// TwinCAT 3 PLC project MachineAlarmManager
// Title: machine_alarm_manager
// Company: Beckhoff Automation K.K.
// Author: Takashi Ichihashi
// ProjectVersion: 1.0.2.0
// ProgramVersion: 3.1.4024.0
// CompilerDefines: VISU_USEWSTRING
// libraries:
//   Tc2_Standard, * (Beckhoff Automation GmbH)
//   Tc2_System, * (Beckhoff Automation GmbH)
//   Tc2_Utilities, * (Beckhoff Automation GmbH)
//   Tc3_EventLogger, * (Beckhoff Automation GmbH)
//   Tc3_Module, * (Beckhoff Automation GmbH)
//   VisuSymbols,3.5.10.0,System
// project tree:
//   DUTs/ AlarmMessage.TcDUT, EventContainer.TcDUT, DataTag.TcDUT, EventActivityFields.TcDUT, EventQueueCommand.TcDUT, EventSeverityStatusMember.TcDUT, EventText.TcDUT, primitives.TcDUT, ST_EventMetadata.TcDUT, ST_EventView.TcDUT, Tc2EventClass.TcDUT, Tc2EventStates.TcDUT
//   / GlobalTextList.TcGTLO, PlcTask.TcTTO, Visualization Manager.TcVMO (not stored), VISU_TASK.TcTTO
//   GVLs/ AlarmEventParam.TcGVL, GVL.TcGVL
//   POUs/ FB_Alarm.TcPOU, FB_EventIoTExporter.TcPOU, FB_EventObserver.TcPOU, FB_Subject.TcPOU, FB_TcEventQueue.TcPOU, FB_Tc3EventVisualizationView.TcPOU, FB_TcEventTable.TcPOU, InterfaceEventViewer.TcIO, AlarmManager.TcPOU, MAIN.TcPOU, UserProgram.TcPOU
//   VISUs/ languages.TcTLO, Visualization.TcVIS, history.TcVIS, current.TcVIS
// real-time tasks:
//   TASK PlcTask: cycle T#10ms, priority 20, ADS port 350
//   TASK VISU_TASK: cycle T#200000us, priority 30, ADS port 351

CONFIGURATION MachineAlarmManager
    RESOURCE PLC ON TwinCAT3
        TASK PlcTask(INTERVAL := T#10ms, PRIORITY := 20);
        TASK VISU_TASK(INTERVAL := T#200000us, PRIORITY := 30);
        PROGRAM MAIN WITH PlcTask : MAIN;
        PROGRAM VisuElems_Visu_Prg WITH VISU_TASK : VisuElems.Visu_Prg;
    END_RESOURCE
END_CONFIGURATION

// ---- DUTs/AlarmMessage.TcDUT
TYPE AlarmMessage EXTENDS EventActivityFields :
STRUCT
	datetime: ULINT;
	sequence_number: ULINT;
END_STRUCT
END_TYPE

// ---- DUTs/EventContainer.TcDUT
TYPE EventContainer :
STRUCT
	event : FB_Alarm;
	{attribute 'TcEncoding' := 'UTF-8'}
	event_text	: T_MaxString;
END_STRUCT
END_TYPE

// ---- DUTs/DataTag.TcDUT
TYPE DataTag :
STRUCT
	{attribute 'TagName' := 'machine_id'}
    machine_id : STRING;
	{attribute 'TagName' := 'module_name'}
    module_name: STRING;
END_STRUCT
END_TYPE

// ---- DUTs/EventActivityFields.TcDUT
TYPE EventActivityFields EXTENDS DataTag:
STRUCT
	{attribute 'TagName' := 'uuid'}
    uuid : STRING;
	{attribute 'FieldName' := 'event_id'}
    event_id : STRING;
	{attribute 'FieldName' := 'severity'}
	severity: INT;
	{attribute 'TcEncoding' := 'UTF-8'}
	{attribute 'FieldName' := 'text'}
    text : STRING;
	{attribute 'FieldName' := 'status'}
    status : BOOL;
END_STRUCT
END_TYPE

// ---- DUTs/EventQueueCommand.TcDUT
TYPE EventQueueCommand :
STRUCT
	metadata : ST_EventMetadata;
	event_text_processor	: FB_RequestEventText;
	event_details_processor	: FB_RequestEventDetails;
END_STRUCT
END_TYPE

// ---- DUTs/EventSeverityStatusMember.TcDUT
TYPE EventSeverityStatusMember :
STRUCT
	severity 	: TcEventSeverity;
	active_counter		: UINT;
	raised_counter		: UINT;
	confirmed_counter	: UINT;
END_STRUCT
END_TYPE

// ---- DUTs/EventText.TcDUT
TYPE EventText :
STRUCT
	event : I_TcEventBase;
	text  : REFERENCE TO STRING;
END_STRUCT
END_TYPE

// ---- DUTs/primitives.TcDUT
TYPE primitives :
UNION
	ARGTYPE_BYTE : BYTE;
    ARGTYPE_WORD : WORD;
    ARGTYPE_DWORD : DWORD;
    ARGTYPE_REAL : REAL;
    ARGTYPE_LREAL : LREAL;
    ARGTYPE_SINT : SINT;
    ARGTYPE_INT : INT;
    ARGTYPE_DINT : DINT;
    ARGTYPE_USINT : USINT;
    ARGTYPE_UINT : UINT;
    ARGTYPE_UDINT : UDINT;
    ARGTYPE_STRING : STRING;
    ARGTYPE_BOOL 	: BOOL;
    ARGTYPE_ULARGE	: ULINT;
    ARGTYPE_UHUGE 	: T_UHUGE_INTEGER;
    ARGTYPE_LARGE	: LINT;
    ARGTYPE_HUGE 	: T_HUGE_INTEGER;
    ARGTYPE_LWORD 	: LWORD;
END_UNION
END_TYPE

// ---- DUTs/ST_EventMetadata.TcDUT
TYPE ST_EventMetadata :
STRUCT
    nEventId          : UDINT;
    eSeverity         : TcEventSeverity;
    bWithConfirmation : BOOL;
	bWithResetOperation : BOOL;
END_STRUCT
END_TYPE

// ---- DUTs/ST_EventView.TcDUT
TYPE ST_EventView :
STRUCT
    nSourceId       : UDINT;
    nEventId        : UDINT;
    Severity        : WSTRING(17);
    ConfirmState   : WSTRING(5);
    sDate           : STRING(23);
    sTime           : STRING(23);
    Computer       : WSTRING;
    sSource         : WSTRING(255);
	MessageText    : WSTRING(255);
    bQuitMessage    : BOOL;
    bConfirmable    : BOOL;
END_STRUCT
END_TYPE

// ---- DUTs/Tc2EventClass.TcDUT
{attribute 'qualified_only'}
{attribute 'strict'}
TYPE Tc2EventClass :
(
	TCEVENTCLASS_NONE := 0,
	TCEVENTCLASS_MAINTENANCE := 1,
	TCEVENTCLASS_MESSAGE :=2,
	TCEVENTCLASS_HINT :=3,
	TCEVENTCLASS_STATEINFO :=4,
	TCEVENTCLASS_INSTRUCTION :=5,
	TCEVENTCLASS_WARNING :=6,
	TCEVENTCLASS_ALARM :=7,
	TCEVENTCLASS_PARAMERROR :=8,
	TCEVENTCLASS_MAX
)DWORD := TCEVENTCLASS_NONE;
END_TYPE

// ---- DUTs/Tc2EventStates.TcDUT
{attribute 'qualified_only'}
{attribute 'strict'}
TYPE Tc2EventStates :
(
	CEVENTSTATE_INVALID := 16#00,
	TCEVENTSTATE_SIGNALED := 16#01,
	TCEVENTSTATE_RESET := 16#02,
	TCEVENTSTATE_CONFIRMED :=16#10,
	TCEVENTSTATE_RESETCON :=16#12
)DWORD;
END_TYPE

// ---- GVLs/AlarmEventParam.TcGVL
{attribute 'qualified_only'}
VAR_GLOBAL CONSTANT
	ALARM_MAX_COUNT: UINT := 3;
END_VAR

// ---- GVLs/GVL.TcGVL
VAR_GLOBAL CONSTANT
	// Database ID
	TARGET_DBID : UINT := 1;
END_VAR
VAR_GLOBAL
	 fb_alarm 		: ARRAY [1..AlarmEventParam.ALARM_MAX_COUNT] OF POINTER TO FB_Alarm;
	 event_initialized	: BOOL;
END_VAR

// ---- POUs/InterfaceEventViewer.TcIO
INTERFACE InterfaceEventViewer

METHOD clear : BOOL
VAR_INPUT
END_VAR
END_METHOD

METHOD history_clear : BOOL
VAR_INPUT
END_VAR
END_METHOD

METHOD send_event : BOOL
VAR_INPUT
	event_container : REFERENCE TO EventContainer;
END_VAR
END_METHOD

METHOD show : BOOL
VAR_INPUT
	event_container : REFERENCE TO EventContainer;
END_VAR
END_METHOD

END_INTERFACE

// ---- POUs/MAIN.TcPOU
PROGRAM MAIN
VAR
END_VAR

AlarmManager();
GVL.event_initialized := AlarmManager.init;
UserProgram();

END_PROGRAM

// ---- POUs/AlarmManager.TcPOU
PROGRAM AlarmManager
VAR_OUTPUT
	init : BOOL;	
END_VAR
VAR
(* Alarm control *)	
	// Alarm calculation function block
	i : UINT;
	
	(*User variables*)
	// User alarm event
	error_condition					: BOOL;
	warning_condition				: BOOL;
	info_condition					: BOOL;

	error_argument				: INT := 0;
	error_code_random			: DRAND; 

	// input FROM HMI
	confirm_button_input		: BOOL;
	reset_button_input			: BOOL;
	history_clear_button_input	: BOOL;
	history_clear_delay_timer	: TON;

	// output to HMI
	status_unconfirm				: BOOL;
	unconfirmed_count				: UDINT;
	status_active					: BOOL;
	active_count					: UDINT;
	status_resetable				: BOOL;
	blink_timer				: TON := (PT := T#0.5S);
	
	(* For Visualization *)
    bReadEvents          : BOOL;
	
	(*Listener*)
	fb_observer : FB_EventObserver;
	subject				: FB_Subject;
	event_table_view 	: FB_Tc3EventVisualizationView;
	event_iot_exporter	: FB_EventIoTExporter;		// IoT exporter
	fbGetTimeZoneInformation	: FB_GetTimeZoneInformation := (bExecute := TRUE);
	
	tmp_string : T_MaxString;
	lang_select_options : UDINT := 1;
	
	alarm_instance : REFERENCE TO FB_ALarm;
	
	(*
	eSeverity ::
	TYPE TcEventSeverity : (
		Verbose  := 0, 
		Info     := 1, 
		Warning  := 2, 
		Error    := 3, 
		Critical := 4);
	END_TYPE
	*)
	AlarmDatabase : ARRAY [1..AlarmEventParam.ALARM_MAX_COUNT] OF ST_EventMetadata := [
		(	
			nEventId := 1,				// イベントID 1 
			eSeverity := 3, 			// TcEventSeverity
			bWithConfirmation := TRUE,	// 新規アラームと確認済みアラームの区別が必要か否か
			bWithResetOperation := TRUE	// アラーム解除のリセット操作が必要か否か
		),
		(	nEventId := 2, 
			eSeverity := 2, 
			bWithConfirmation := TRUE,
			bWithResetOperation := FALSE
		),
		(	nEventId := 3, 
			eSeverity := 1, 
			bWithConfirmation := FALSE,
			bWithResetOperation := TRUE
		)
	];
END_VAR

(*
	FB_Observer内の FB_Alarm インスタンス配列に対して、GVL.AlarmDatabseで定義したイベントクラスの情報で紐付ける。
*)
IF NOT init THEN
	FOR i := 1 TO AlarmEventParam.ALARM_MAX_COUNT DO
		fb_observer.event_table.init_instance(
			eventClass := TC_EVENT_CLASSES.UserEventClass,
			nEventId := AlarmDatabase[i].nEventId,
			eSeverity := AlarmDatabase[i].eSeverity,
			bWithConfirmation := AlarmDatabase[i].bWithConfirmation,
			bWithResetOperation := AlarmDatabase[i].bWithResetOperation
		);
		alarm_instance REF= fb_observer.event_table.get_alarm(i);
		GVL.fb_alarm[i] := ADR(alarm_instance);
	END_FOR
	fb_observer.event_table.viewer := subject;
	subject.subscribe(event_table_view);
	subject.subscribe(event_iot_exporter);
	init := TRUE;
END_IF

//　アラームリセットボタン受付
IF reset_button_input THEN
	fb_observer.event_table.try_clear_all_alarm();
END_IF

// アラーム確認ボタン受付
IF confirm_button_input THEN
	fb_observer.event_table.confirm_all_alarm();
END_IF


// IPCのロケール設定の読み出しと、Visualization向けイベントテーブル表示FBへのタイムゾーン情報設定
IF fbGetTimeZoneInformation.bBusy THEN
	fbGetTimeZoneInformation.bExecute := FALSE;		
END_IF
fbGetTimeZoneInformation();
event_table_view.tzinfo := fbGetTimeZoneInformation.tzInfo;
event_iot_exporter.tzinfo := fbGetTimeZoneInformation.tzInfo;

// オブザーバ（監視）オブジェクトの実行
CASE lang_select_options OF
	0: fb_observer.nLangId := 1033;
	1: fb_observer.nLangId := 1041;
END_CASE
fb_observer(event_class := TC_EVENT_CLASSES.UserEventClass);

// 表示用の変数制御　（アクティブアラーム数、未確認アラーム数、ボタン点滅制御、リセット可能状態）
active_count := fb_observer.event_table.active_event_count;
status_active := active_count > 0;
unconfirmed_count := fb_observer.event_table.unconfirmed_event_count;

status_resetable := fb_observer.event_table.set_event_count = 0 AND status_active;

IF unconfirmed_count > 0 THEN
	blink_timer(IN := NOT blink_timer.Q);
	IF blink_timer.Q THEN
		status_unconfirm := NOT status_unconfirm;
	END_IF
ELSE
	status_unconfirm := status_active;
END_IF

// 履歴の消去(5秒長押し）
history_clear_delay_timer(IN := history_clear_button_input, PT := T#5S);
IF history_clear_delay_timer.Q THEN
	fb_observer.event_table.viewer.history_clear();
END_IF

END_PROGRAM

// ---- POUs/FB_EventObserver.TcPOU
FUNCTION_BLOCK FB_EventObserver EXTENDS FB_ListenerBase2
VAR_INPUT
	event_class : GUID;
	nLangId		: DINT := 1033;
	subscribe : BOOL := TRUE;
END_VAR
VAR_OUTPUT
	subscribed	: BOOL;
END_VAR
VAR
	i : UDINT;
	fbListenerFilter : FB_TcEventFilter; 
	active_alarm_count : UDINT;
	_queue	: FB_TcEventQueue;
	_event_table : FB_TcEventTable;
	init :BOOL;
END_VAR

_queue.nLangId := nLangId;

IF NOT init THEN
	_event_table.queue REF= _queue;
	init := TRUE;
END_IF

IF subscribe AND NOT THIS^.bSubscribed THEN 
	fbListenerFilter.Clear().EventClass.EqualTo(event_class); //define all events (messages and alarms) from this eventclass   
	THIS^.Subscribe2(fbListenerFilter); //subscribe to retrieve defined events
END_IF

IF event_class.DATA1 <> 0 THEN
	_event_table.event_class := event_class;
END_IF

IF NOT subscribe AND THIS^.bSubscribed THEN 
	THIS^.Unsubscribe();
END_IF 

subscribed := THIS^.bSubscribed;
THIS^.Execute();
_event_table();

PROPERTY event_table : REFERENCE TO FB_TcEventTable
GET
event_table REF= _event_table;
END_GET
END_PROPERTY

METHOD OnAlarmCleared : HRESULT
VAR_INPUT
	fbEvent : REFERENCE TO FB_TcEvent;
END_VAR
VAR
END_VAR
_event_table.remove_event(fbEvent);
_event_table.create_view();
OnAlarmCleared := S_OK;
END_METHOD

METHOD OnAlarmConfirmed : HRESULT
VAR_INPUT
	fbEvent : REFERENCE TO FB_TcEvent;
END_VAR
_event_table.create_view();
OnAlarmConfirmed := S_OK;
END_METHOD

METHOD OnAlarmRaised : HRESULT
VAR_INPUT
	fbEvent : REFERENCE TO FB_TcEvent;
END_VAR
VAR
	_request_text 	: REFERENCE TO FB_RequestEventText;
END_VAR
_event_table.add_event(fbEvent);
_queue.put(fbEvent);
OnAlarmRaised := S_OK;
END_METHOD

METHOD OnMessageSent : HRESULT
VAR_INPUT
	fbEvent : REFERENCE TO FB_TcEvent;
END_VAR
OnMessageSent := S_OK;
END_METHOD

END_FUNCTION_BLOCK

// ---- POUs/FB_TcEventQueue.TcPOU
FUNCTION_BLOCK FB_TcEventQueue
VAR CONSTANT
	COMMAND_QUEUE_BUFFER_SIZE :UDINT := 20;
END_VAR
VAR_INPUT
	nLangId : DINT := 1033;
END_VAR
VAR_OUTPUT
END_VAR
VAR
	_usage:	UDINT;
	_write_index : UDINT := 1;
	_read_index : UDINT := 1;
	_queue_size:	UDINT := COMMAND_QUEUE_BUFFER_SIZE;
	queue_buffer:	ARRAY [1..COMMAND_QUEUE_BUFFER_SIZE] OF EventQueueCommand;
END_VAR

PROPERTY full : BOOL
GET
full :=  _usage >= COMMAND_QUEUE_BUFFER_SIZE;
END_GET
END_PROPERTY

METHOD get : REFERENCE TO EventQueueCommand
VAR_INPUT
END_VAR
IF _usage = 0 THEN
	get REF= 0;
	RETURN;
END_IF

get REF= queue_buffer[_read_index];

_usage := _usage - 1;

IF COMMAND_QUEUE_BUFFER_SIZE > _read_index THEN
	_read_index := _read_index + 1;
ELSE
	_read_index := 1;
END_IF
END_METHOD

METHOD put : BOOL
VAR_INPUT
	fbEvent:	REFERENCE TO FB_TcEvent;
END_VAR
IF _usage >= COMMAND_QUEUE_BUFFER_SIZE THEN
	put := FALSE;
ELSE
	queue_buffer[_write_index].metadata.bWithConfirmation := FALSE;
	queue_buffer[_write_index].metadata.eSeverity := fbEvent.eSeverity;
	queue_buffer[_write_index].metadata.nEventId := fbEvent.nEventId;
	queue_buffer[_write_index].event_text_processor.Request(
				eventClass := fbEvent.EventClass, 
				nEventId := fbEvent.nEventId, 
				nLangId := nLangId, 
				ipArgs := fbEvent.ipArguments
			);

	_usage := _usage + 1;
	IF COMMAND_QUEUE_BUFFER_SIZE > _write_index THEN
		_write_index := _write_index + 1;
	ELSE
		_write_index := 1;
	END_IF
	put := TRUE;
END_IF
END_METHOD

PROPERTY usage : UDINT
GET
usage := _usage;
END_GET
END_PROPERTY

END_FUNCTION_BLOCK

// ---- POUs/FB_TcEventTable.TcPOU
FUNCTION_BLOCK FB_TcEventTable
VAR CONSTANT
	EVENT_INDEX_TABLE_SIZE : UDINT := 80;
END_VAR
VAR_INPUT
END_VAR
VAR_OUTPUT
END_VAR
VAR
	i : UDINT;
	init : BOOL;
	_queue : REFERENCE TO FB_TcEventQueue;
	_viewer : InterfaceEventViewer;
	_metadata : REFERENCE TO EventQueueCommand;
	_p_alarm	: POINTER TO FB_TcAlarm;
	_event_class	: GUID;
	_unconfirmed_event_count : UDINT;
	_active_event_count : UDINT;
	_set_event_count	: UDINT;
	await : BOOL;
	event_max_index : UDINT := 0;
	event_table  : ARRAY [1..AlarmEventParam.ALARM_MAX_COUNT] OF EventContainer;
	active_event_table	: ARRAY [1..EVENT_INDEX_TABLE_SIZE] OF POINTER TO EventContainer;
	active_event_max_index	: UDINT := 1;

	target_active_index : UDINT := 1;
	target_event_index : UDINT := 1;	
	view_refresh_flag : BOOL;
	
	view_terminate : BOOL;

	current_event : REFERENCE TO FB_Alarm;
END_VAR

// Getting text asynchronous process
IF NOT await AND _queue.usage > 0 THEN
	_metadata REF= _queue.get();
	IF __ISVALIDREF(_metadata) THEN
		await := TRUE;
	END_IF
END_IF



IF await THEN
	target_active_index := get_active_event_by_id(GUID_TO_STRING(_event_class), _metadata.metadata.nEventId);
	IF target_active_index <> 0 THEN
		IF _metadata.event_text_processor.GetString(
				active_event_table[target_active_index]^.event_text,
				SIZEOF(active_event_table[target_active_index]^.event_text)
		) THEN
			_viewer.send_event(active_event_table[target_active_index]^);
			create_view();
			await := FALSE;
		END_IF
	END_IF
END_IF

// Continuous execution for each event
REPEAT
	current_event REF= iter();
	IF __ISVALIDREF(current_event) THEN
		current_event();
	END_IF
UNTIL 
	NOT __ISVALIDREF(current_event)
END_REPEAT

// Refresh current aram list view
IF view_refresh_flag THEN
	_unconfirmed_event_count := 0;
	_active_event_count := 0;
	_viewer.clear(); // Once clear whole of items.
	i := 1;
	REPEAT
		IF i <= active_event_max_index THEN
			IF active_event_table[i] <> 0 THEN
				view_terminate := _viewer.show(active_event_table[i]^);
				_active_event_count := _active_event_count + 1;
				IF active_event_table[i]^.event.eConfirmationState = TcEventConfirmationState.WaitForConfirmation THEN
					_unconfirmed_event_count := _unconfirmed_event_count + 1;
				END_IF
			END_IF
		END_IF
		i := i + 1;
	UNTIL
		i > active_event_max_index OR view_terminate
	END_REPEAT
	view_refresh_flag := FALSE;
END_IF

// Watch every time.
_set_event_count := 0;
i := 1;
REPEAT
	IF i <= active_event_max_index AND active_event_table[i] <> 0 THEN
		IF active_event_table[i]^.event.set_activate THEN
			_set_event_count := _set_event_count + 1;
		END_IF
	END_IF
	i := i + 1;
UNTIL
	i > active_event_max_index
END_REPEAT

PROPERTY active_event_count : UDINT
GET
active_event_count := _active_event_count;
END_GET
END_PROPERTY

METHOD add_event : BOOL
VAR_INPUT
	fbEvent	: REFERENCE TO FB_TcEvent;
END_VAR
VAR
	active_index 	: UDINT;
	event_index 	: UDINT;
	first_null_index		: UDINT;
END_VAR
event_index := get_event_by_event(fbEvent);
first_null_index := 0;
FOR active_index := 1 TO active_event_max_index DO
	IF active_event_table[active_index] = 0 THEN
		IF first_null_index = 0 THEN
			first_null_index := active_index;
		END_IF
	ELSIF ADR(event_table[event_index]) = active_event_table[active_index] THEN
		RETURN;
	END_IF
END_FOR

IF first_null_index = 0 THEN
	active_event_max_index := active_index;
ELSE
	active_index := first_null_index;
END_IF

active_event_table[active_index] := ADR(event_table[event_index]);
END_METHOD

METHOD confirm_all_alarm : BOOL
VAR_INPUT
END_VAR
FOR i := 1 TO event_max_index DO
	event_table[i].event.set_confirm := TRUE;
END_FOR
END_METHOD

METHOD create_view : BOOL
VAR_INPUT
END_VAR
VAR
	i : UDINT;
END_VAR
IF _viewer <> 0 THEN
	view_refresh_flag := TRUE;
END_IF
END_METHOD

PROPERTY event_class : GUID
SET
_event_class := event_class;
END_SET
END_PROPERTY

METHOD get_active_event_by_id : UDINT
VAR_INPUT
	sEventClass	: STRING;
	nEventID	: UDINT;
END_VAR
VAR
	i : UDINT;
END_VAR
get_active_event_by_id := 0;

FOR i := 1 TO active_event_max_index DO
	IF active_event_table[i] <> 0 THEN
		IF GUID_TO_STRING(active_event_table[i]^.event.EventClass) = sEventClass AND active_event_table[i]^.event.nEventId = nEventID THEN
			get_active_event_by_id := i;
			RETURN;
		END_IF		
	END_IF
END_FOR
END_METHOD

METHOD get_alarm : REFERENCE TO FB_Alarm
VAR_INPUT
	index : UDINT;
END_VAR
IF index <= event_max_index THEN
	get_alarm REF= event_table[index].event;
ELSE
	get_alarm REF= 0;
END_IF
END_METHOD

METHOD get_event_by_event : UDINT
VAR_INPUT
	event	: I_TcEventBase;
END_VAR
VAR
	i : UDINT;
END_VAR
get_event_by_event := 0;

FOR i := 1 TO event_max_index DO
	IF event_table[i].event.EqualsTo(event) THEN
		get_event_by_event := i;
		RETURN;
	END_IF
END_FOR
END_METHOD

METHOD init_instance : POINTER TO FB_Alarm
VAR_INPUT
	eventClass			: GUID; // イベントクラスのGUID
	nEventId			: UDINT; // 登録したイベントID
	eSeverity			: TcEventSeverity; // 重要度
	bWithConfirmation	: BOOL;
	bWithResetOperation	: BOOL;
END_VAR
IF event_max_index >= AlarmEventParam.ALARM_MAX_COUNT THEN
	init_instance := 0;
	RETURN;
END_IF

event_max_index := event_max_index + 1;
event_table[event_max_index].event.Create(
			eventClass := eventClass,
			nEventId := nEventId,
			eSeverity := eSeverity,
			bWithConfirmation := bWithConfirmation,
			ipSourceInfo := 0
		);
event_table[event_max_index].event.bWithResetOperation := bWithResetOperation;

init_instance := ADR(event_table[event_max_index]);
END_METHOD

METHOD iter : REFERENCE TO FB_Alarm
VAR_INPUT
END_VAR
VAR_INST
	last_index : UDINT := 1;
END_VAR
VAR
	i : UDINT;
END_VAR
IF last_index > event_max_index THEN
	iter REF= 0;
	last_index := 1;
ELSE
	iter REF= event_table[last_index].event;
	last_index := last_index + 1;
END_IF
END_METHOD

PROPERTY queue : REFERENCE TO FB_TcEventQueue
SET
_queue REF= queue;
END_SET
END_PROPERTY

METHOD remove_event : BOOL
VAR_INPUT
	fbEvent	: REFERENCE TO FB_TcEvent;
END_VAR
VAR
	active_index 	: UDINT;
	last_active_index	: UDINT;
	
END_VAR
VAR_INST
	not_found_error: BOOL;
END_VAR
not_found_error := TRUE;
FOR active_index := 1 TO active_event_max_index DO
	IF active_event_table[active_index] <> 0 THEN
		IF active_event_table[active_index]^.event.EqualsTo(fbEvent) THEN
			_viewer.send_event(active_event_table[active_index]^);
			active_event_table[active_index] := 0;
			IF active_index = active_event_max_index THEN
				active_event_max_index := last_active_index;
			END_IF
		END_IF
		not_found_error := FALSE;
		last_active_index := active_index;
	END_IF
END_FOR

remove_event := NOT not_found_error;
END_METHOD

PROPERTY set_event_count : UDINT
GET
set_event_count := _set_event_count;
END_GET
END_PROPERTY

METHOD try_clear_all_alarm : BOOL
VAR_INPUT
END_VAR
VAR
END_VAR
FOR i := 1 TO event_max_index DO
	event_table[i].event.set_clear := TRUE;
END_FOR
END_METHOD

PROPERTY unconfirmed_event_count : UDINT
GET
unconfirmed_event_count := _unconfirmed_event_count;
END_GET
END_PROPERTY

PROPERTY viewer : InterfaceEventViewer
GET
viewer := _viewer;
END_GET
SET
_viewer := viewer;
END_SET
END_PROPERTY

END_FUNCTION_BLOCK

// ---- POUs/FB_Alarm.TcPOU
FUNCTION_BLOCK FB_Alarm EXTENDS FB_TcAlarm
VAR_INPUT
	set_activate	: BOOL;				// Set true during something event occured.
	set_confirm		: BOOL;				// True momentally after operator confirming event.
	set_clear		: BOOL := FALSE;	// When the bLatch flag is True and bEvt is False, this flag can be unlatch when raised. 
	module_name 	:STRING;			// module name where event occured.
	nLangId			: DINT := 1033;		// Language code
END_VAR
VAR
	set_activate_mem	: BOOL;				// Set true during something event occured.	
	_with_reset_operation : BOOL;
END_VAR
VAR PERSISTENT
	_sequence_number	: ULINT;	
END_VAR

IF set_activate  
	AND NOT SUPER^.bRaised AND
	SUPER^.eConfirmationState <> TcEventConfirmationState.WaitForConfirmation THEN
	SUPER^.Raise(0);
	SUPER^.ipArguments.Clear();
END_IF

IF set_confirm THEN
	SUPER^.Confirm(0);
END_IF


//IF SUPER^.eConfirmationState = TcEventConfirmationState.NotSupported THEN
IF NOT _with_reset_operation THEN
	IF set_activate_mem AND NOT set_activate THEN
		SUPER^.Clear(0, TRUE);
	END_IF
ELSE
	IF NOT set_activate 
		AND set_clear THEN
		SUPER^.Clear(0, TRUE);
	END_IF
END_IF

set_activate_mem	:= set_activate;
set_clear := FALSE;
set_confirm := FALSE;

METHOD add_arguments : BOOL
VAR_INPUT
	argument_value : T_Arg;
END_VAR
VAR
	_temp : primitives;
END_VAR
add_arguments := TRUE;
CASE argument_value.eType OF
    E_ArgType.ARGTYPE_BYTE:
		MEMCPY(ADR(_temp.ARGTYPE_BYTE), argument_value.pData, argument_value.cbLen);
		SUPER^.ipArguments.AddByte(_temp.ARGTYPE_BYTE);
    E_ArgType.ARGTYPE_WORD:
		MEMCPY(ADR(_temp.ARGTYPE_WORD), argument_value.pData, argument_value.cbLen);
		SUPER^.ipArguments.AddWord(_temp.ARGTYPE_WORD);
    E_ArgType.ARGTYPE_DWORD:
		MEMCPY(ADR(_temp.ARGTYPE_DWORD), argument_value.pData, argument_value.cbLen);
		SUPER^.ipArguments.AddDWord(_temp.ARGTYPE_DWORD);
    E_ArgType.ARGTYPE_REAL:
		MEMCPY(ADR(_temp.ARGTYPE_REAL), argument_value.pData, argument_value.cbLen);
		SUPER^.ipArguments.AddReal(_temp.ARGTYPE_REAL);
    E_ArgType.ARGTYPE_LREAL:
		MEMCPY(ADR(_temp.ARGTYPE_LREAL), argument_value.pData, argument_value.cbLen);
		SUPER^.ipArguments.AddLreal(_temp.ARGTYPE_LREAL);
    E_ArgType.ARGTYPE_SINT:
		MEMCPY(ADR(_temp.ARGTYPE_SINT), argument_value.pData, argument_value.cbLen);
		SUPER^.ipArguments.AddSint(_temp.ARGTYPE_SINT);
    E_ArgType.ARGTYPE_INT:
		MEMCPY(ADR(_temp.ARGTYPE_INT), argument_value.pData, argument_value.cbLen);
		SUPER^.ipArguments.AddInt(_temp.ARGTYPE_INT);
    E_ArgType.ARGTYPE_DINT:
		MEMCPY(ADR(_temp.ARGTYPE_DINT), argument_value.pData, argument_value.cbLen);
		SUPER^.ipArguments.AddDint(_temp.ARGTYPE_DINT);
    E_ArgType.ARGTYPE_USINT:
		MEMCPY(ADR(_temp.ARGTYPE_USINT), argument_value.pData, argument_value.cbLen);
		SUPER^.ipArguments.AddUsint(_temp.ARGTYPE_USINT);
    E_ArgType.ARGTYPE_UINT:
		MEMCPY(ADR(_temp.ARGTYPE_UINT), argument_value.pData, argument_value.cbLen);
		SUPER^.ipArguments.AddUint(_temp.ARGTYPE_UINT);
    E_ArgType.ARGTYPE_UDINT:
		MEMCPY(ADR(_temp.ARGTYPE_UDINT), argument_value.pData, argument_value.cbLen);
		SUPER^.ipArguments.AddUdint(_temp.ARGTYPE_UDINT);
    E_ArgType.ARGTYPE_STRING:
		MEMCPY(ADR(_temp.ARGTYPE_STRING), argument_value.pData, argument_value.cbLen);
		SUPER^.ipArguments.AddString(_temp.ARGTYPE_STRING);
    E_ArgType.ARGTYPE_BOOL:
		MEMCPY(ADR(_temp.ARGTYPE_BOOL), argument_value.pData, argument_value.cbLen);
		SUPER^.ipArguments.AddBool(_temp.ARGTYPE_BOOL);
    E_ArgType.ARGTYPE_ULARGE:
		MEMCPY(ADR(_temp.ARGTYPE_ULARGE), argument_value.pData, argument_value.cbLen);
		SUPER^.ipArguments.AddULInt(_temp.ARGTYPE_ULARGE);
    E_ArgType.ARGTYPE_LARGE:
		MEMCPY(ADR(_temp.ARGTYPE_LARGE), argument_value.pData, argument_value.cbLen);
		SUPER^.ipArguments.AddLint(_temp.ARGTYPE_LARGE);
	ELSE
		add_arguments := FALSE;
END_CASE
END_METHOD

PROPERTY bWithResetOperation : BOOL
GET
bWithResetOperation := _with_reset_operation;
END_GET
SET
_with_reset_operation := bWithResetOperation;
END_SET
END_PROPERTY

END_FUNCTION_BLOCK

// ---- POUs/FB_Subject.TcPOU
FUNCTION_BLOCK FB_Subject IMPLEMENTS InterfaceEventViewer
VAR CONSTANT
	MAX_EVENTS : UDINT := 10;
END_VAR
VAR
	event_containers	: ARRAY [1..MAX_EVENTS] OF InterfaceEventViewer;
	max_index			: UDINT;
END_VAR

{warning 'add method implementation '}
METHOD clear : BOOL
VAR
	i : UDINT;
END_VAR
FOR i := 1 TO max_index DO
	IF event_containers[i] <> 0 THEN
		event_containers[i].clear();
	END_IF
END_FOR
END_METHOD

{warning 'add method implementation '}
METHOD history_clear : BOOL
VAR
	i : UDINT;
END_VAR
FOR i := 1 TO max_index DO
	IF event_containers[i] <> 0 THEN
		event_containers[i].history_clear();
	END_IF
END_FOR
END_METHOD

{warning 'add method implementation '}
METHOD send_event : BOOL
VAR_INPUT
	event_container	: REFERENCE TO EventContainer;
END_VAR
VAR
	i : UDINT;
END_VAR
FOR i := 1 TO max_index DO
	IF event_containers[i] <> 0 THEN
		event_containers[i].send_event(event_container);
	END_IF
END_FOR
END_METHOD

{warning 'add method implementation '}
METHOD show : BOOL
VAR_INPUT
	event_container	: REFERENCE TO EventContainer;
END_VAR
VAR
	i : UDINT;
END_VAR
FOR i := 1 TO max_index DO
	IF event_containers[i] <> 0 THEN
		event_containers[i].show(event_container);
	END_IF
END_FOR
END_METHOD

METHOD subscribe : UDINT
VAR_INPUT
	observable	: InterfaceEventViewer;
END_VAR
VAR
	i : UDINT;
END_VAR
subscribe := 0;
FOR i := 1 TO MAX_EVENTS DO
	IF event_containers[i] = 0 THEN
		event_containers[i] := observable;
		IF i > max_index THEN
			max_index := i;
		END_IF
		subscribe := i;
		RETURN;
	END_IF
END_FOR
END_METHOD

METHOD unsubscribe : BOOL
VAR_INPUT
	subscriber : UDINT;
END_VAR
VAR
	i : UDINT;
END_VAR
IF event_containers[subscriber] <> 0 THEN
	event_containers[subscriber] := 0;
	IF subscriber = max_index THEN
		FOR i := max_index TO 0 BY -1 DO
			IF event_containers[i] <> 0 THEN
				max_index := 1;
			END_IF
		END_FOR
	END_IF
	unsubscribe := TRUE;
ELSE
	unsubscribe := FALSE;
END_IF
END_METHOD

END_FUNCTION_BLOCK

// ---- POUs/FB_Tc3EventVisualizationView.TcPOU
FUNCTION_BLOCK FB_Tc3EventVisualizationView IMPLEMENTS InterfaceEventViewer
VAR CONSTANT
	DISP_ROWS : UDINT := 80;
END_VAR
VAR_INPUT
	tzinfo : ST_TimeZoneInformation;
END_VAR
VAR_OUTPUT PERSISTENT
	stAlarmEvents	: ARRAY [1..DISP_ROWS] OF ST_EventView;
	stAlarmhistory 	: ARRAY [1..DISP_ROWS] OF ST_EventView;
END_VAR
VAR
	row : UDINT := 1;
END_VAR

METHOD PRIVATE _create_current_table : BOOL
VAR_INPUT
	event_container : REFERENCE TO EventContainer;
	row		: UDINT;
	stDate	: STRING;
	stTime	: STRING;
END_VAR
VAR
	iso_datetime : STRING;
	source_name : STRING;
END_VAR
UTF8_TO_WSTRING(
	ADR(stAlarmEvents[row].Computer),
	ADR(event_container.event.module_name),
	SIZEOF(stAlarmEvents[row].Computer)
);

source_name := event_container.event.ipSourceInfo.sName;

UTF8_TO_WSTRING(
	ADR(stAlarmEvents[row].sSource),
	ADR(source_name),
	SIZEOF(stAlarmEvents[row].sSource)
);

stAlarmEvents[row].bConfirmable := event_container.event.eConfirmationState <> TcEventConfirmationState.NotSupported;
CASE event_container.event.eSeverity OF 
	TcEventSeverity.Critical:
		stAlarmEvents[row].Severity := "危険";		
	TcEventSeverity.Error:
		stAlarmEvents[row].Severity := "異常";
	TcEventSeverity.Info:
		stAlarmEvents[row].Severity := "情報";
	TcEventSeverity.Verbose:
		stAlarmEvents[row].Severity := "ログ";
	TcEventSeverity.Warning:
		stAlarmEvents[row].Severity := "警告";
	ELSE
		stAlarmEvents[row].Severity := TO_WSTRING(event_container.event.eSeverity);
END_CASE

CASE event_container.event.eConfirmationState OF 
	TcEventConfirmationState.Confirmed:
		stAlarmEvents[row].ConfirmState := "レ";
	TcEventConfirmationState.WaitForConfirmation:
		stAlarmEvents[row].ConfirmState := "";
	ELSE
		stAlarmEvents[row].ConfirmState := "--";
END_CASE

stAlarmEvents[row].nEventId := event_container.event.nEventId;
UTF8_TO_WSTRING(
	ADR(stAlarmEvents[row].MessageText),
	ADR(event_container.event_text),
	SIZEOF(stAlarmEvents[row].MessageText)
);


iso_datetime := FILETIME64_TO_ISO8601(
					fileTime := event_container.event.nTimeRaised,
					nBias := TO_INT(tzInfo.bias), 
					bUTC :=TRUE, 
					nPrecision := 0
				);
stAlarmEvents[row].sDate := MID(iso_datetime, 10, 1);
stAlarmEvents[row].sTime := MID(iso_datetime, 8, 12);
END_METHOD

METHOD clear : BOOL
row := 1;
MEMSET(ADR(stAlarmEvents), 0, SIZEOF(stAlarmEvents));
END_METHOD

{warning 'add method implementation '}
METHOD history_clear : BOOL
MEMSET(ADR(stAlarmhistory), 0, SIZEOF(stAlarmhistory));
END_METHOD

METHOD send_event : BOOL
VAR_INPUT
	event_container	: REFERENCE TO EventContainer;
END_VAR
VAR
	iso_datetime : STRING;
	source_name : STRING;
END_VAR
MEMMOVE(ADR(stAlarmhistory[2]), ADR(stAlarmhistory[1]), ADR(stAlarmhistory[DISP_ROWS - 1]) - ADR(stAlarmhistory[1]));

UTF8_TO_WSTRING(
	ADR(stAlarmhistory[1].Computer),
	ADR(event_container.event.module_name),
	SIZEOF(stAlarmhistory[1].Computer)
);

source_name := event_container.event.ipSourceInfo.sName;

UTF8_TO_WSTRING(
	ADR(stAlarmhistory[1].sSource),
	ADR(source_name),
	SIZEOF(stAlarmhistory[1].sSource)
);

stAlarmhistory[1].bConfirmable := event_container.event.eConfirmationState <> TcEventConfirmationState.NotSupported;
CASE event_container.event.eSeverity OF 
	TcEventSeverity.Critical:
		stAlarmhistory[1].Severity := "危険";		
	TcEventSeverity.Error:
		stAlarmhistory[1].Severity := "異常";
	TcEventSeverity.Info:
		stAlarmhistory[1].Severity := "情報";
	TcEventSeverity.Verbose:
		stAlarmhistory[1].Severity := "ログ";
	TcEventSeverity.Warning:
		stAlarmhistory[1].Severity := "警告";
	ELSE
		stAlarmhistory[1].Severity := TO_WSTRING(event_container.event.eSeverity);
END_CASE

IF event_container.event.bRaised THEN 
	stAlarmhistory[1].ConfirmState := "発生";
ELSE
	stAlarmhistory[1].ConfirmState := "解除";
END_IF

stAlarmhistory[1].nEventId := event_container.event.nEventId;
UTF8_TO_WSTRING(
	ADR(stAlarmhistory[1].MessageText),
	ADR(event_container.event_text),
	SIZEOF(stAlarmhistory[1].MessageText)
);


IF event_container.event.bRaised THEN
	iso_datetime := FILETIME64_TO_ISO8601(
						fileTime := event_container.event.nTimeRaised,
						nBias := TO_INT(tzInfo.bias), 
						bUTC :=TRUE, 
						nPrecision := 0
					);
ELSE
	iso_datetime := FILETIME64_TO_ISO8601(
						fileTime := event_container.event.nTimeCleared,
						nBias := TO_INT(tzInfo.bias), 
						bUTC :=TRUE, 
						nPrecision := 0
					);	
END_IF

stAlarmhistory[1].sDate := MID(iso_datetime, 10, 1);
stAlarmhistory[1].sTime := MID(iso_datetime, 8, 12);
END_METHOD

METHOD show : BOOL
VAR_INPUT
	event_container : REFERENCE TO EventContainer;
END_VAR
VAR_INST
	iso_datetime : STRING;
END_VAR
VAR
	stDate	: STRING;
	stTime	: STRING;
END_VAR
IF NOT __ISVALIDREF(event_container) OR row > DISP_ROWS THEN
	show := TRUE;
	RETURN;
END_IF

iso_datetime := FILETIME64_TO_ISO8601(
					fileTime := event_container.event.nTimeRaised,
					nBias := TO_INT(tzInfo.bias), 
					bUTC :=TRUE, 
					nPrecision := 0
				);

stDate := MID(iso_datetime, 10, 1);
stTime := MID(iso_datetime, 8, 12);

_create_current_table(event_container, row, stDate, stTime);
			
row := row + 1;
show := FALSE;
END_METHOD

END_FUNCTION_BLOCK

// ---- POUs/FB_EventIoTExporter.TcPOU
FUNCTION_BLOCK FB_EventIoTExporter IMPLEMENTS InterfaceEventViewer
VAR_INPUT
	tzinfo : ST_TimeZoneInformation;
END_VAR
VAR_OUTPUT
	export_event : ST_EventView;
END_VAR
VAR
END_VAR

{warning 'add method implementation '}
METHOD clear : BOOL
END_METHOD

{warning 'add method implementation '}
METHOD history_clear : BOOL
END_METHOD

{warning 'add method implementation '}
METHOD send_event : BOOL
VAR_INPUT
	event_container	: REFERENCE TO EventContainer;
END_VAR
VAR
	iso_datetime : STRING;
	source_name : STRING;
END_VAR
IF event_container.event.bRaised THEN
	UTF8_TO_WSTRING(
		ADR(export_event.Computer),
		ADR(event_container.event.module_name),
		SIZEOF(export_event.Computer)
	);
	
	source_name := event_container.event.ipSourceInfo.sName;
	
	UTF8_TO_WSTRING(
		ADR(export_event.sSource),
		ADR(source_name),
		SIZEOF(export_event.sSource)
	);
	
	export_event.bConfirmable := event_container.event.eConfirmationState <> TcEventConfirmationState.NotSupported;
	CASE event_container.event.eSeverity OF 
		TcEventSeverity.Critical:
			export_event.Severity := "危険";		
		TcEventSeverity.Error:
			export_event.Severity := "異常";
		TcEventSeverity.Info:
			export_event.Severity := "情報";
		TcEventSeverity.Verbose:
			export_event.Severity := "ログ";
		TcEventSeverity.Warning:
			export_event.Severity := "警告";
		ELSE
			export_event.Severity := TO_WSTRING(event_container.event.eSeverity);
	END_CASE
	
	IF event_container.event.bRaised THEN 
		export_event.ConfirmState := "発生";
	ELSE
		export_event.ConfirmState := "解除";
	END_IF
	
	export_event.nEventId := event_container.event.nEventId;
	UTF8_TO_WSTRING(
		ADR(export_event.MessageText),
		ADR(event_container.event_text),
		SIZEOF(export_event.MessageText)
	);
	
	
	IF event_container.event.bRaised THEN
		iso_datetime := FILETIME64_TO_ISO8601(
							fileTime := event_container.event.nTimeRaised,
							nBias := TO_INT(tzInfo.bias), 
							bUTC :=TRUE, 
							nPrecision := 0
						);
	ELSE
		iso_datetime := FILETIME64_TO_ISO8601(
							fileTime := event_container.event.nTimeCleared,
							nBias := TO_INT(tzInfo.bias), 
							bUTC :=TRUE, 
							nPrecision := 0
						);	
	END_IF
	
	export_event.sDate := MID(iso_datetime, 10, 1);
	export_event.sTime := MID(iso_datetime, 8, 12);
END_IF
END_METHOD

{warning 'add method implementation '}
METHOD show : BOOL
VAR_INPUT
	event_container	: REFERENCE TO EventContainer;
END_VAR
END_METHOD

END_FUNCTION_BLOCK

// ---- POUs/UserProgram.TcPOU
PROGRAM UserProgram
VAR
	// input FROM HMI
	is_error					: BOOL;
	is_warning					: BOOL;
	is_info						: BOOL;
	
	error_argument				: INT := 0;
	error_code_random			: DRAND; 
	tmp_string 					: STRING(255);
END_VAR

// Simply set "GVL.fb_alarm[*]^.set_activate" true when alarm is activated.
// 

IF GVL.event_initialized THEN
	// アラーム1　（Alarmレベル） 発報制御
	IF is_error THEN												// is_errorが エラー状態 bit
		error_code_random(Seed := 1);
		error_argument := TO_INT(error_code_random.Num * 32767.0);	// 疑似的に乱数によりエラーコードを生成
		GVL.fb_alarm[1]^.ipArguments.Clear();							// Event Class に登録したEventのDisplay text の {0} {1} に展開した文字をクリアにする。
		tmp_string := 'Error Code';									// F_STRING() の引数は VAR_IN_OUT なのでリテラルは使えない。一旦仮変数にセットする。
		GVL.fb_alarm[1]^.add_arguments(F_STRING(tmp_string));			// Event Class に登録したEventのDisplay text の {0} 部分に埋め込まれる値。 T_Arg型でセット。
		GVL.fb_alarm[1]^.add_arguments(F_Int(error_argument));		// Event Class に登録したEventのDisplay text の {1} 部分に埋め込まれる値。 T_Arg型でセット。
	END_IF
	GVL.fb_alarm[1]^.set_activate := is_error;						// エラー状態の通知。エラーテキストに　{0} や {1} などの付加的な情報が無ければこの 1 行だけで良い。
	
	// アラーム2　（Warningレベル） 発報制御
	IF is_warning THEN
		error_code_random(Seed := 1);
		error_argument := TO_INT(error_code_random.Num * 32767.0);
		GVL.fb_alarm[2]^.ipArguments.Clear();
		tmp_string := 'Warning Code';	
		GVL.fb_alarm[2]^.add_arguments(F_STRING(tmp_string));
		GVL.fb_alarm[2]^.add_arguments(F_Int(error_argument));
	END_IF
	GVL.fb_alarm[2]^.set_activate := is_warning;
	
	
	// アラーム3　（Informationレベル） 発報制御
	IF is_info THEN
		error_code_random(Seed := 1);
		error_argument := TO_INT(error_code_random.Num * 32767.0);
		GVL.fb_alarm[3]^.ipArguments.Clear();
		tmp_string := 'Status';
		GVL.fb_alarm[3]^.add_arguments(F_STRING(tmp_string));
		GVL.fb_alarm[3]^.add_arguments(F_Int(error_argument));
	END_IF
	GVL.fb_alarm[3]^.set_activate := is_info;
END_IF

END_PROGRAM

// ---- GlobalTextList.TcGTLO
TEXTLIST GlobalTextList
  206 = '%S'
  174 = '%s'
  15 = 'AlarmManager.event_table_view.stAlarmEvents[INDEX].Computer'
  562 = 'Critical'
  870 = 'Critical\n発報'
  436 = 'Errorレベル'
  513 = 'Errorレベル\n以上'
  401 = 'Errorレベル以上'
  30 = 'ID'
  715 = 'Info\n発報'
  924 = 'Infoレベル'
  413 = 'Infoレベル\n以上'
  351 = 'MAIN.event_table_view.stAlarmEvents[INDEX].Severity'
  571 = 'MessageText'
  639 = 'tesut'
  71 = 'Warning\n発報'
  682 = 'Warningレベル'
  725 = 'Warningレベル\n以上'
  324 = 'アラーム'
  283 = 'テキスト'
  486 = 'リセット'
  854 = '内容'
  814 = '履歴'
  714 = '履歴消去'
  601 = '日付'
  947 = '時刻'
  945 = '未確認アラーム数'
  105 = '現在'
  655 = '発生中アラーム数'
  902 = '確認'
  819 = '言語設定'
  136 = '重要度'
END_TEXTLIST

// ---- VISUs/languages.TcTLO
TEXTLIST languages
  0 = '英語'
  1 = '日本語'
   = ''
END_TEXTLIST

// ---- VISUs/Visualization.TcVIS
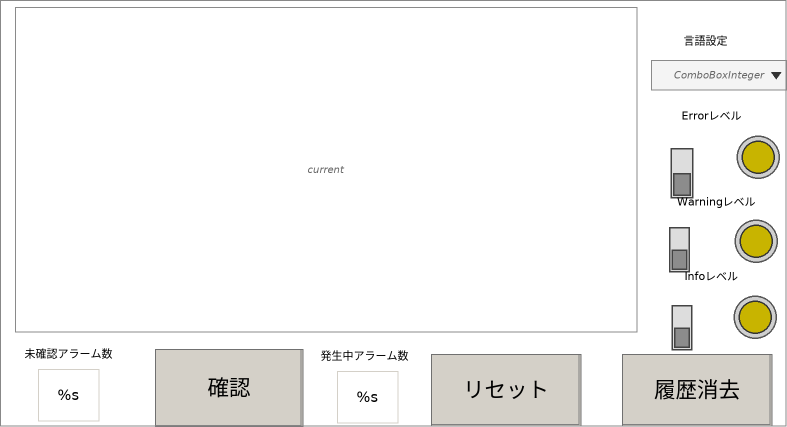
VISUALIZATION Visualization  // 787x427
    Button (155,349 148x78), "確認", colour toggle: AlarmManager.status_unconfirm, pressed state: AlarmManager.confirm_button_input
        tap AlarmManager.confirm_button_input
    DipSwitch (657,145 50x56), variable: UserProgram.is_error, behaviour: TOGGLE, style: Switch-DipSwitch-Gray
    Button (431,354 150x72), "リセット", colour toggle: AlarmManager.status_resetable, pressed state: AlarmManager.reset_button_input
        tap AlarmManager.reset_button_input
    DipSwitch (656,227 47x45), variable: UserProgram.is_warning, behaviour: TOGGLE, style: Switch-DipSwitch-Gray
    DipSwitch (656,305 52x45), variable: UserProgram.is_info, behaviour: TOGGLE, style: Switch-DipSwitch-Gray
    Lamp1 (733,131 50x52), variable: UserProgram.is_error, style: Lamp-Lamp1-Yellow
    Lamp1 (731,215 50x52), variable: UserProgram.is_warning, style: Lamp-Lamp1-Yellow
    Lamp1 (730,291 50x52), variable: UserProgram.is_info, style: Lamp-Lamp1-Yellow
    Label (670,99 83x34), "Errorレベル"
    Label (675,185 83x34), "Warningレベル"
    Label (670,265 83x23), "Infoレベル"
    Textfield (38,369 61x52), "%s", text variable: AlarmManager.unconfirmed_count
    Textfield (337,371 61x52), "%s", text variable: AlarmManager.active_count
    Label (308,341 113x30), "発生中アラーム数"
    Label (12,339 113x30), "未確認アラーム数"
    TabControl (15,7 622x325)
        shows current()
        shows history()
        [0]: TabTitle=現在
        [1]: TabTitle=履歴
    Label (664,24 83x34), "言語設定"
    ComboBoxInteger (651,60 136x30), variable: AlarmManager.lang_select_options, text list: 'languages'
    Button (622,354 150x72), "履歴消去"
        tap AlarmManager.history_clear_button_input
END_VISUALIZATION

// ---- VISUs/history.TcVIS
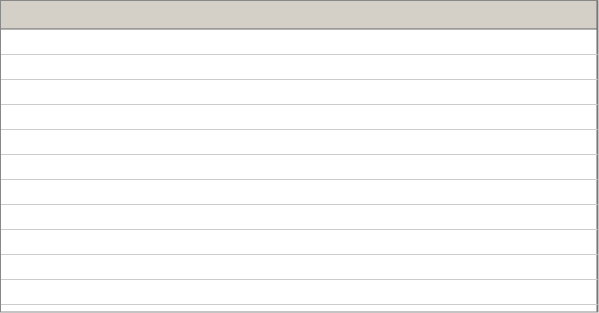
VISUALIZATION history  // 599x313
    Table (-2,-1 599x313), data array: AlarmManager.event_table_view.stAlarmhistory
        p3854506369: AlarmManager.event_table_view.stAlarmhistory[INDEX].nSourceId
        p1892666644: AlarmManager.event_table_view.stAlarmhistory[INDEX].nEventId
        p338671338: AlarmManager.event_table_view.stAlarmhistory[INDEX].Severity
        p2170511999: AlarmManager.event_table_view.stAlarmhistory[INDEX].ConfirmState
        p3723444502: AlarmManager.event_table_view.stAlarmhistory[INDEX].sDate
        p1218418051: AlarmManager.event_table_view.stAlarmhistory[INDEX].sTime
        p746581629: AlarmManager.event_table_view.stAlarmhistory[INDEX].Computer
        p3104783080: AlarmManager.event_table_view.stAlarmhistory[INDEX].sSource
        p2501879983: AlarmManager.event_table_view.stAlarmhistory[INDEX].MessageText
        p7306298: AlarmManager.event_table_view.stAlarmhistory[INDEX].bQuitMessage
        p1933151965: AlarmManager.event_table_view.stAlarmhistory[INDEX].bConfirmable
        p1755163831: 重要度
        p4092479075: 履歴
        p2237128397: 日付
        p505689113: 時刻
        p2243050616: テキスト
END_VISUALIZATION

// ---- VISUs/current.TcVIS
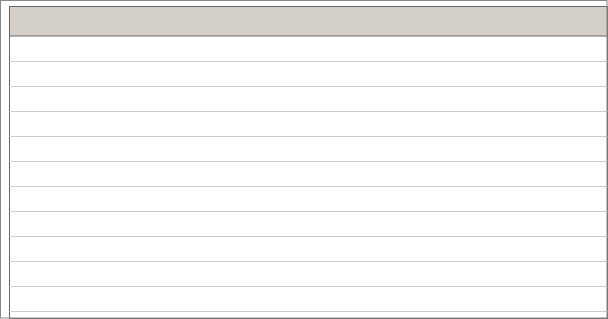
VISUALIZATION current  // 608x319
    Table (9,6 599x313), data array: AlarmManager.event_table_view.stAlarmEvents
        p3854506369: AlarmManager.event_table_view.stAlarmEvents[INDEX].nSourceId
        p1892666644: AlarmManager.event_table_view.stAlarmEvents[INDEX].nEventId
        p338671338: AlarmManager.event_table_view.stAlarmEvents[INDEX].Severity
        p2170511999: AlarmManager.event_table_view.stAlarmEvents[INDEX].ConfirmState
        p3723444502: AlarmManager.event_table_view.stAlarmEvents[INDEX].sDate
        p1218418051: AlarmManager.event_table_view.stAlarmEvents[INDEX].sTime
        p746581629: AlarmManager.event_table_view.stAlarmEvents[INDEX].Computer
        p3104783080: AlarmManager.event_table_view.stAlarmEvents[INDEX].sSource
        p2501879983: AlarmManager.event_table_view.stAlarmEvents[INDEX].MessageText
        p7306298: AlarmManager.event_table_view.stAlarmEvents[INDEX].bQuitMessage
        p1933151965: AlarmManager.event_table_view.stAlarmEvents[INDEX].bConfirmable
        p1755163831: 重要度
        p4092479075: 確認
        p2237128397: 日付
        p505689113: 時刻
        p2243050616: テキスト
END_VISUALIZATION
